// TIA Portal project "Connection" (V17)

(* hardware
DEVICE "S7-1500/ET200MP station_1"  S7-1500 station
   slot 0: "Rail_0"  Rack  6ES7 590-1***0-0AA0
   slot 1: "PLC_1"  CPU 1515-2 PN  6ES7 515-2AM02-0AB0  V2.9
      slot 3: "CPU display_1"  6ES7591-1BA00-0AA0
      slot 32768: "PROFINET interface_1"  X1
         slot 32769: "Port_1"  X1 P1
         slot 32770: "Port_2"  X1 P2
      slot 33024: "PROFINET interface_2"  X2
         slot 33025: "Port_1"  X2 P1
      slot 34817: "Virtual CP interface port_1"  Virtual CP interface port  Virtual CP interface port
*)

// ===== PLC "PLC_1"  CPU 1515-2 PN =====

VAR_GLOBAL   // PLC tag table "Default tag table"
   "Tag_1" AT %M50.0 : Bool;
   "Tag_2" AT %M50.1 : Bool;
   "opc_t1" AT %IW100 : Int;
END_VAR

DATA_BLOCK "ModbusConn"   // DB2
{ S7_Optimized_Access := 'FALSE' }
VERSION : 0.1
   VAR
      Connection : TCON_IP_v4;
      Connection_1 : TCON_IP_v4;
   END_VAR
BEGIN
   Connection.RemoteAddress.ADDR[1] := 195;
   Connection.RemoteAddress.ADDR[2] := 168;
   Connection.RemoteAddress.ADDR[3] := 0;
   Connection.RemoteAddress.ADDR[4] := 5;
   Connection.RemotePort := 0;
   Connection.InterfaceId := 64;
   Connection.ID := 1;
   Connection.ConnectionType := 11;
   Connection.ActiveEstablished := false;
   Connection.LocalPort := 502;
   Connection_1.InterfaceId := 64;
   Connection_1.ID := 2;
   Connection_1.ConnectionType := 11;
   Connection_1.ActiveEstablished := false;
   Connection_1.RemoteAddress.ADDR[1] := 195;
   Connection_1.RemoteAddress.ADDR[2] := 168;
   Connection_1.RemoteAddress.ADDR[3] := 0;
   Connection_1.RemoteAddress.ADDR[4] := 5;
   Connection_1.RemotePort := 0;
   Connection_1.LocalPort := 502;
END_DATA_BLOCK

DATA_BLOCK "ModbusData"   // DB3
{ S7_Optimized_Access := 'FALSE' }
VERSION : 0.1
   VAR
      HoldingRegister : Array[0..30] of Word;
   END_VAR
BEGIN
END_DATA_BLOCK

DATA_BLOCK "Modbus_Bool"   // DB4
{ S7_Optimized_Access := 'FALSE' }
VERSION : 0.1
   VAR
      Boolean : Array[0..30] of Bool;
   END_VAR
BEGIN
END_DATA_BLOCK

DATA_BLOCK "opc_data"   // DB5
{ S7_Optimized_Access := 'FALSE' }
VERSION : 0.1
   VAR
      "Server interface_1.TEST_OPC.data1" : Int;
      "Server interface_1.TEST_OPC.data2" : Int;
      "Server interface_1.TEST_OPC.data3" : Int;
      "Server interface_1.TEST_OPC.data4" : Int;
      "Server interface_1.TEST_OPC.data5" : Int;
      "Server interface_1.TEST_OPC.data6" : Int;
      "Server interface_1.TEST_OPC.data7" : Int;
      "Server interface_1.TEST_OPC.data8" : Int;
      "Server interface_1.TEST_OPC.data9" : Int;
      "Server interface_1.TEST_OPC.data10" : Int;
      "Server interface_1.TEST_OPC.data11" : Int;
      "Server interface_1.TEST_OPC.data12" : Int;
      "Server interface_1.TEST_OPC.data13" : Int;
      "Server interface_1.TEST_OPC.data14" : Int;
      "Server interface_1.TEST_OPC.data15" : Int;
      "Server interface_1.TEST_OPC.data16" : Int;
      "Server interface_1.TEST_OPC.data17" : Int;
      "Server interface_1.TEST_OPC.data18" : Int;
      "Server interface_1.TEST_OPC.data19" : Int;
      "Server interface_1.TEST_OPC.data20" : Int;
      "Server interface_1.TEST_OPC.data21" : Int;
      "Server interface_1.TEST_OPC.data22" : Int;
      "Server interface_1.TEST_OPC.data23" : Int;
      "Server interface_1.TEST_OPC.data24" : Int;
      "Server interface_1.TEST_OPC.data25" : Int;
      "Server interface_1.TEST_OPC.data26" : Int;
      "Server interface_1.TEST_OPC.data27" : Int;
      "Server interface_1.TEST_OPC.data28" : Bool;
      "Server interface_1.TEST_OPC.data29" : Bool;
      "Server interface_1.TEST_OPC.data30" : Bool;
      "Server interface_1.TEST_OPC.data31" : Bool;
      "Server interface_1.TEST_OPC.data32" : Bool;
      "Server interface_1.TEST_OPC.data33" : Bool;
      "Server interface_1.TEST_OPC.data34" : Bool;
      "Server interface_1.TEST_OPC.data35" : Bool;
      "Server interface_1.TEST_OPC.data36" : Bool;
      "Server interface_1.TEST_OPC.Static.data1" : Int;
   END_VAR
BEGIN
END_DATA_BLOCK

DATA_BLOCK "Profinet_Conn"   // DB100
{ S7_Optimized_Access := 'FALSE' }
VERSION : 0.1
   VAR
      word1 : Word;
      word2 : Word;
      word3 : Word;
      word4 : Word;
      word5 : Word;
      word6 : Word;
      word7 : Word;
      word8 : Word;
      word9 : Word;
      int1 : Int;
      int2 : Int;
      int3 : Int;
      int4 : Int;
      int5 : Int;
      int6 : Int;
      int7 : Int;
      int8 : Int;
      int9 : Int;
      real1 : Real;
      real2 : Real;
      real3 : Real;
      real4 : Real;
      real5 : Real;
      real6 : Real;
      real7 : Real;
      real8 : Real;
      real9 : Real;
      bool1 : Bool;
      bool2 : Bool;
      bool3 : Bool;
      bool4 : Bool;
      bool5 : Bool;
      bool6 : Bool;
      bool7 : Bool;
      bool8 : Bool;
      bool9 : Bool;
   END_VAR
BEGIN
END_DATA_BLOCK

ORGANIZATION_BLOCK "Main"   // OB1, LAD, ProgramCycle
TITLE = "Main Program Sweep (Cycle)"
{ S7_Optimized_Access := 'TRUE' }
VERSION : 0.1
   VAR_INPUT
      Initial_Call : Bool;   // Initial call of this OB
      Remanence : Bool;   // =True, if remanent data are available
   END_VAR
BEGIN

REGION Network 1
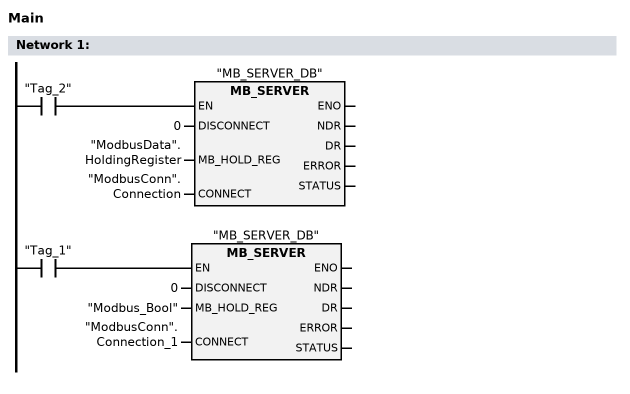
   IF "Tag_2" THEN
       "MB_SERVER_DB"(DISCONNECT := 0,   // MB_SERVER
                      MB_HOLD_REG := "ModbusData".HoldingRegister,
                      CONNECT := "ModbusConn".Connection);
   END_IF;
   IF "Tag_1" THEN
       "MB_SERVER_DB"(DISCONNECT := 0, MB_HOLD_REG := "Modbus_Bool", CONNECT := "ModbusConn".Connection_1);   // MB_SERVER
   END_IF;
END_REGION
END_ORGANIZATION_BLOCK